(* IEC 61131-3 sources: mastertool-rankine-bridge/tests/indexer/fixtures/sample_export/objects/application_fb_1__FB_Malformado, 1 file *)

(* ---- declaration.st ---- *)
FUNCTION_BLOCK FB_Malformado
VAR_INPUT
    xEntrada        : BOOL;
VAR_OUTPUT
    xSaida          : BOOL;
END_VAR
